// TIA Portal project "dec_to_bin" (V14)

(* hardware
DEVICE "S7-1200 station_1"  S7-1200 Station
   slot 0: "Rack_0"  S7-1200 Rack  Rack  V1.0
   slot 1: "PLC_1"  CPU 1214C DC/DC/DC  6ES7 214-1AG40-0XB0  V4.2
*)

// ===== PLC "PLC_1"  CPU 1214C DC/DC/DC =====

VAR_GLOBAL   // PLC tag table "Default tag table"
   "B_" AT %I0.0 : Bool;
   "A__" AT %I0.1 : Bool;
   "Tag_1" AT %Q0.1 : Bool;
   "Tag_2" AT %Q0.0 : Bool;
   "Tag_3" AT %IW64 : Word;
   "Tag_4" AT %MD10 : Real;
   "Tag_5" AT %MD14 : DWord;
   "Tag_6" AT %I0.3 : Bool;
   "Tag_7" AT %I0.5 : Bool;
   "Tag_8" AT %I0.7 : Bool;
   "Tag_9" AT %I0.2 : Bool;
   "Tag_10" AT %I0.6 : Bool;
   "Tag_11" AT %I0.4 : Bool;
   "tmp1" AT %M0.0 : Bool;
   "tmp2" AT %M0.1 : Bool;
   "tmp3" AT %M0.2 : Bool;
   "Tag_12" AT %Q0.2 : Bool;
END_VAR

ORGANIZATION_BLOCK "Main"   // OB1, LAD, ProgramCycle
TITLE = "Main Program Sweep (Cycle)"
{ S7_Optimized_Access := 'TRUE' }
VERSION : 0.1
   VAR_INPUT
      Initial_Call : Bool;   // Initial call of this OB
      Remanence : Bool;   // =True, if remanent data are available
   END_VAR
   VAR_TEMP
      A_ : Bool;
   END_VAR
BEGIN

REGION Network 1
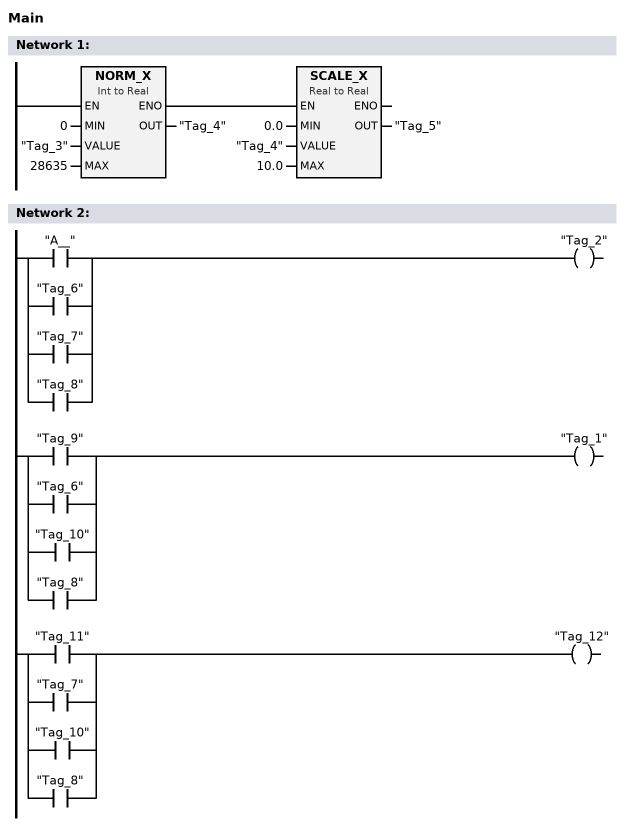
   RUNG wire#powerrail
      { S7_Templates := "[SrcType := Int, DestType := Real]" } Normalize(min := 0, value := "Tag_3", max := 28635, out => "Tag_4")
      { S7_Templates := "[SrcType := Real, DestType := Real]" } Scale(min := 0.0, value := "Tag_4", max := 10.0, out => "Tag_5")
   END_RUNG
   // the same network as SCL:
   "Tag_4" := NORM_X(MIN := 0, VALUE := "Tag_3", MAX := 28635);
   "Tag_5" := SCALE_X(MIN := 0.0, VALUE := "Tag_4", MAX := 10.0);
END_REGION

REGION Network 2
   RUNG wire#powerrail
      Contact( "A__" )
      wire#w1
      Coil( "Tag_2" )
   END_RUNG
   RUNG wire#powerrail
      Contact( "Tag_6" )
   END_RUNG wire#w1
   RUNG wire#powerrail
      Contact( "Tag_7" )
   END_RUNG wire#w1
   RUNG wire#powerrail
      Contact( "Tag_8" )
   END_RUNG wire#w1
   RUNG wire#powerrail
      Contact( "Tag_9" )
      wire#w2
      Coil( "Tag_1" )
   END_RUNG
   RUNG wire#powerrail
      Contact( "Tag_6" )
   END_RUNG wire#w2
   RUNG wire#powerrail
      Contact( "Tag_10" )
   END_RUNG wire#w2
   RUNG wire#powerrail
      Contact( "Tag_8" )
   END_RUNG wire#w2
   RUNG wire#powerrail
      Contact( "Tag_11" )
      wire#w3
      Coil( "Tag_12" )
   END_RUNG
   RUNG wire#powerrail
      Contact( "Tag_7" )
   END_RUNG wire#w3
   RUNG wire#powerrail
      Contact( "Tag_10" )
   END_RUNG wire#w3
   RUNG wire#powerrail
      Contact( "Tag_8" )
   END_RUNG wire#w3
   // the same network as SCL:
   "Tag_2" := "A__" OR "Tag_6" OR "Tag_7" OR "Tag_8";
   "Tag_1" := "Tag_9" OR "Tag_6" OR "Tag_10" OR "Tag_8";
   "Tag_12" := "Tag_11" OR "Tag_7" OR "Tag_10" OR "Tag_8";
END_REGION
END_ORGANIZATION_BLOCK